FOR _idx := 0 TO RobotLibraryParameter.SUB_PROGRAM_DATA_MAX
DO
  // add command.Data[_idx]
  CreateCommandPayload.AddByte(_command.Data[_idx]);
END_FOR

// Create logging
CreateCommandPayloadLog(AxesGroup := AxesGroup);
END_METHOD

METHOD INTERNAL CreateCommandPayloadLog
VAR_IN_OUT
  /// Robot assignment of function
  AxesGroup : AxesGroup; 
END_VAR
VAR
  /// internal index for loops
 _idx : DINT;
END_VAR
// Create log entry for Parameter start
CreateLogMessage      ( Timestamp   := AxesGroup.InternalData.SystemTime,
                        MessageType := MessageType.CMD,
                        Severity    := Severity.DEBUG,
                        MessageCode := 0,
                        MessageText := 'Create command payload with the following parameter(s) :');
  
// Create log entry for EmitterID[x]
FOR _idx := 0 TO 3
DO
  CreateLogMessagePara2 ( Timestamp   := AxesGroup.InternalData.SystemTime,
                          MessageType := MessageType.CMD,
                          Severity    := Severity.DEBUG,
                          MessageCode := 0,
                          MessageText := 'Command.EmitterID[{2}] = {1}',
                          Para1       :=  SINT_TO_STRING(_command.EmitterID[_idx]),
                          Para2       :=  DINT_TO_STRING(_idx));
END_FOR

// Create log entry for ListenerID
CreateLogMessagePara1 ( Timestamp   := AxesGroup.InternalData.SystemTime,
                        MessageType := MessageType.CMD,
                        Severity    := Severity.DEBUG,
                        MessageCode := 0,
                        MessageText := 'Command.ListenerID = {1}',
                        Para1       :=  SINT_TO_STRING(_command.ListenerID));

// Create log entry for Reserve
CreateLogMessagePara1 ( Timestamp   := AxesGroup.InternalData.SystemTime,
                        MessageType := MessageType.CMD,
                        Severity    := Severity.DEBUG,
                        MessageCode := 0,
                        MessageText := 'Command.Reserve = {1}',
                        Para1       :=  BYTE_TO_STRING(_command.Reserve));

// Create log entry for JobID
CreateLogMessagePara1 ( Timestamp   := AxesGroup.InternalData.SystemTime,
                        MessageType := MessageType.CMD,
                        Severity    := Severity.DEBUG,
                        MessageCode := 0,
                        MessageText := 'Command.JobID = {1}',
                        Para1       :=  UINT_TO_STRING(_command.JobID));

FOR _idx := 0 TO RobotLibraryParameter.SUB_PROGRAM_DATA_MAX
DO
  // Create log entry for Data
  CreateLogMessagePara1 ( Timestamp   := AxesGroup.InternalData.SystemTime,
                          MessageType := MessageType.CMD,
                          Severity    := Severity.DEBUG,
                          MessageCode := 0,
                          MessageText := StrReplace('Command.Data[{0}] = {1}', '{0}', DINT_TO_STRING(_idx)), 
                          Para1       :=  UINT_TO_STRING(_command.Data[_idx]));
END_FOR
END_METHOD

METHOD FB_init : BOOL
VAR_INPUT
  /// if TRUE, the retain variables are initialized (warm start / cold start)
  bInitRetains : BOOL; 
  /// if TRUE, the instance afterwards gets moved into the copy code (online change)
  bInCopyCode  : BOOL;  
END_VAR
MyType := 'MC_CallSubprogramFB';

ExecMode := ExecutionMode.PARALLEL;
END_METHOD

METHOD PROTECTED OnCall
VAR_IN_OUT
  /// Robot assignment of function
  AxesGroup : AxesGroup; 
END_VAR
// call base implementation
SUPER^.OnCall(AxesGroup := AxesGroup);

CASE _stepCmd OF
  
  00:  IF ( _execute_R.Q )  
       THEN
         // Check function is supported and parameter are valid ?
         IF (( CheckFunctionSupported( AxesGroup := AxesGroup )) AND
             ( CheckParameterValid   ( AxesGroup := AxesGroup )))      
         THEN
           // set busy flag
           Busy := TRUE;
           // Reset command outputs
           SysDepMemSet(pDest := ADR(OutCmd), Value := 0, DataLen := SIZEOF(OutCmd));         
           // apply command parameter
          _parCmd := ParCmd;
           // init parameter sequence
          _command.ParSeq := 1;
           // create command data
           CommandData := CreateCommandPayload(AxesGroup := AxesGroup);
           // Add command to active command register
          _uniqueID := AxesGroup.Acyclic.ActiveCommandRegister.AddCmd( pCommandFB := ADR(THIS^ ));     
           // set timeout
           SetTimeout(PT := _timeoutCmd, rTimer := _timerCmd);
           // inc step counter
          _stepCmd := _stepCmd + 1; 
          END_IF
       END_IF
     

  01:  // Wait for responce received
       IF ( _responseReceived )
       THEN
         // reset response received flag
        _responseReceived := FALSE;

         CASE  _response.State 
         OF
           CmdMessageState.BUFFERED    : CommandBuffered    := TRUE;
           CmdMessageState.INTERRUPTED : CommandInterrupted := TRUE;           
           CmdMessageState.DONE        : Done               := TRUE;           
           CmdMessageState.ABORTED     : CommandAborted     := TRUE;
           CmdMessageState.ERROR       : Error              := TRUE;
         END_CASE
                
         InProgress := _response.InProgress;
         
         // Done, Aborted or Error ?
         IF (_response.State >= CmdMessageState.DONE )
         THEN
           // reset Busy flag
           Busy := FALSE;
           // Update results
           OutCmd.InstanceID        := 0; {warning 'ToDo'}
           OutCmd.OriginID          := _response.OriginID;
           OutCmd.InvocationCounter := _response.InvocationCounter;
           OutCmd.ReturnData        := _response.ReturnData;
 
           // set timeout
           SetTimeout(PT := _timeoutCmd, rTimer := _timerCmd);
           // inc step counter
          _stepCmd := _stepCmd + 1; 
         END_IF
       END_IF


  02: IF ( NOT Execute)
      THEN
        Reset();
      END_IF     
ELSE
  // invalid step
  ErrorID := RobotLibraryEvents.ERR_INVALID_STEP;
END_CASE



// Reset FB
IF ( NOT Execute )
THEN
  Reset();  
END_IF
END_METHOD

METHOD INTERNAL ParseResponsePayload : DINT
VAR_INPUT
  /// Response data
  ResponseData : RobotLibraryRecvDataFB;
  /// Timestamp
  Timestamp    : SystemTime;  
END_VAR
VAR
  /// internal index for loops
 _idx : DINT;
END_VAR

// Table 6-688: Received CMD payload (RC to PLC) of "CallSubprogram"
// --------------------------
// Header
// --------------------------
// Byte 00 : USINT   - ParSeq | State     
// Byte 01 : SINT    - AlarmMessageSeverity    
// Byte 02 : UINT    - AlarmMessageCode HB
// Byte 03 :         - AlarmMessageCode LB
// --------------------------
// Datablock
// --------------------------
// Byte 04 : USINT InvocationCounter;
// Byte 05 : SINT  Reserved;
// Byte 06 : INT   OriginID;
// Byte 07 :       OriginID;
// Byte 08 : UINT  Progress;
// Byte 09 :       Progress;
// Byte 10 : BOOL  InProgress;
// Byte 11 : BYTE  ReturnData[0];
// Byte 12 : BYTE  ReturnData[1];
// Byte 13 : BYTE  ReturnData[2];
// Byte 14 : BYTE  ReturnData[3];
// Byte 15 : BYTE  ReturnData[4];
// Byte 16 : BYTE  ReturnData[5];
// Byte 17 : BYTE  ReturnData[6];
// Byte 18 : BYTE  ReturnData[7];
// Byte 19 : BYTE  ReturnData[8];
// Byte 20 : BYTE  ReturnData[9];
// Byte 21 : BYTE  ReturnData[10];
// Byte 22 : BYTE  ReturnData[11];
// Byte 23 : BYTE  ReturnData[12];
// Byte 24 : BYTE  ReturnData[13];
// Byte 25 : BYTE  ReturnData[14];
// Byte 26 : BYTE  ReturnData[15];
// Byte 27 : BYTE  ReturnData[16];
// Byte 28 : BYTE  ReturnData[17];
// Byte 29 : BYTE  ReturnData[18];
// Byte 30 : BYTE  ReturnData[19];
// Byte 31 : BYTE  ReturnData[20];
// Byte 32 : BYTE  ReturnData[21];
// Byte 33 : BYTE  ReturnData[22];
// Byte 34 : BYTE  ReturnData[23];
// Byte 35 : BYTE  ReturnData[24];
// Byte 36 : BYTE  ReturnData[25];
// Byte 37 : BYTE  ReturnData[26];
// Byte 38 : BYTE  ReturnData[27];
// Byte 39 : BYTE  ReturnData[28];
// Byte 40 : BYTE  ReturnData[29];
// Byte 41 : BYTE  ReturnData[30];
// Byte 42 : BYTE  ReturnData[31];
// Byte 43 : BYTE  ReturnData[32];
// Byte 44 : BYTE  ReturnData[33];
// Byte 45 : BYTE  ReturnData[34];
// Byte 46 : BYTE  ReturnData[35];
// Byte 47 : BYTE  ReturnData[36];
// Byte 48 : BYTE  ReturnData[37];
// Byte 49 : BYTE  ReturnData[38];
// Byte 50 : BYTE  ReturnData[39];
// Byte 51 : BYTE  ReturnData[40];
// Byte 52 : BYTE  ReturnData[41];
// Byte 53 : BYTE  ReturnData[42];
// Byte 54 : BYTE  ReturnData[43];
// Byte 55 : BYTE  ReturnData[44];
// Byte 56 : BYTE  ReturnData[45];
// Byte 57 : BYTE  ReturnData[46];
// Byte 58 : BYTE  ReturnData[47];
// Byte 59 : BYTE  ReturnData[48];
// Byte 60 : BYTE  ReturnData[49];
// Byte 61 : BYTE  ReturnData[50];
// Byte 62 : BYTE  ReturnData[51];
// Byte 63 : BYTE  ReturnData[52];
// Byte 64 : BYTE  ReturnData[53];
// Byte 65 : BYTE  ReturnData[54];
// Byte 66 : BYTE  ReturnData[55];
// Byte 67 : BYTE  ReturnData[56];
// Byte 68 : BYTE  ReturnData[57];
// Byte 69 : BYTE  ReturnData[58];
// Byte 70 : BYTE  ReturnData[59];
// Byte 71 : BYTE  ReturnData[60];
// Byte 72 : BYTE  ReturnData[61];
// Byte 73 : BYTE  ReturnData[62];
// Byte 74 : BYTE  ReturnData[63];
// Byte 75 : BYTE  ReturnData[64];
// Byte 76 : BYTE  ReturnData[65];
// Byte 77 : BYTE  ReturnData[66];
// Byte 78 : BYTE  ReturnData[67];
// Byte 79 : BYTE  ReturnData[68];
// Byte 80 : BYTE  ReturnData[69];
// Byte 81 : BYTE  ReturnData[70];
// Byte 82 : BYTE  ReturnData[71];
// Byte 83 : BYTE  ReturnData[72];
// Byte 84 : BYTE  ReturnData[73];
// Byte 85 : BYTE  ReturnData[74];
// Byte 86 : BYTE  ReturnData[75];
// Byte 87 : BYTE  ReturnData[76];
// Byte 88 : BYTE  ReturnData[77];
// Byte 89 : BYTE  ReturnData[78];
// Byte 90 : BYTE  ReturnData[79];
// Byte 91 : BYTE  ReturnData[80];
// Byte 92 : BYTE  ReturnData[81];
// Byte 93 : BYTE  ReturnData[82];
// Byte 94 : BYTE  ReturnData[83];
// Byte 95 : BYTE  ReturnData[84];
// Byte 96 : BYTE  ReturnData[85];
// Byte 97 : BYTE  ReturnData[86];
// Byte 98 : BYTE  ReturnData[87];
// Byte 99 : BYTE  ReturnData[88];
// Byte 100: BYTE  ReturnData[89];
// Byte 101: BYTE  ReturnData[90];
// Byte 102: BYTE  ReturnData[91];
// Byte 103: BYTE  ReturnData[92];
// Byte 104: BYTE  ReturnData[93];
// Byte 105: BYTE  ReturnData[94];
// Byte 106: BYTE  ReturnData[95];
// Byte 107: BYTE  ReturnData[96];
// Byte 108: BYTE  ReturnData[97];
// Byte 109: BYTE  ReturnData[98];
// Byte 110: BYTE  ReturnData[99];
// Byte 111: BYTE  ReturnData[100];
// Byte 112: BYTE  ReturnData[101];
// Byte 113: BYTE  ReturnData[102];
// Byte 114: BYTE  ReturnData[103];
// Byte 115: BYTE  ReturnData[104];
// Byte 116: BYTE  ReturnData[105];
// Byte 117: BYTE  ReturnData[106];
// Byte 118: BYTE  ReturnData[107];
// Byte 119: BYTE  ReturnData[108];
// Byte 120: BYTE  ReturnData[109];
// Byte 121: BYTE  ReturnData[110];
// Byte 122: BYTE  ReturnData[111];
// Byte 123: BYTE  ReturnData[112];
// Byte 124: BYTE  ReturnData[113];
// Byte 125: BYTE  ReturnData[114];
// Byte 126: BYTE  ReturnData[115];
// Byte 127: BYTE  ReturnData[116];
// Byte 128: BYTE  ReturnData[117];
// Byte 129: BYTE  ReturnData[118];
// Byte 130: BYTE  ReturnData[119];
// Byte 131: BYTE  ReturnData[120];
// Byte 132: BYTE  ReturnData[121];
// Byte 133: BYTE  ReturnData[122];
// Byte 134: BYTE  ReturnData[123];
// Byte 135: BYTE  ReturnData[124];
// Byte 136: BYTE  ReturnData[125];
// Byte 137: BYTE  ReturnData[126];
// Byte 138: BYTE  ReturnData[127];
// Byte 139: BYTE  ReturnData[128];
// Byte 140: BYTE  ReturnData[129];
// Byte 141: BYTE  ReturnData[130];
// Byte 142: BYTE  ReturnData[131];
// Byte 143: BYTE  ReturnData[132];
// Byte 144: BYTE  ReturnData[133];
// Byte 145: BYTE  ReturnData[134];
// Byte 146: BYTE  ReturnData[135];
// Byte 147: BYTE  ReturnData[136];
// Byte 148: BYTE  ReturnData[137];
// Byte 149: BYTE  ReturnData[138];
// Byte 150: BYTE  ReturnData[139];
// Byte 151: BYTE  ReturnData[140];
// Byte 152: BYTE  ReturnData[141];
// Byte 153: BYTE  ReturnData[142];
// Byte 154: BYTE  ReturnData[143];
// Byte 155: BYTE  ReturnData[144];
// Byte 156: BYTE  ReturnData[145];
// Byte 157: BYTE  ReturnData[146];
// Byte 158: BYTE  ReturnData[147];
// Byte 159: BYTE  ReturnData[148];
// Byte 160: BYTE  ReturnData[149];
// Byte 161: BYTE  ReturnData[150];
// Byte 162: BYTE  ReturnData[151];
// Byte 163: BYTE  ReturnData[152];
// Byte 164: BYTE  ReturnData[153];
// Byte 165: BYTE  ReturnData[154];
// Byte 166: BYTE  ReturnData[155];
// Byte 167: BYTE  ReturnData[156];
// Byte 168: BYTE  ReturnData[157];
// Byte 169: BYTE  ReturnData[158];
// Byte 170: BYTE  ReturnData[159];
// Byte 171: BYTE  ReturnData[160];
// Byte 172: BYTE  ReturnData[161];
// Byte 173: BYTE  ReturnData[162];
// Byte 174: BYTE  ReturnData[163];
// Byte 175: BYTE  ReturnData[164];
// Byte 176: BYTE  ReturnData[165];
// Byte 177: BYTE  ReturnData[166];
// Byte 178: BYTE  ReturnData[167];
// Byte 179: BYTE  ReturnData[168];
// Byte 180: BYTE  ReturnData[169];
// Byte 181: BYTE  ReturnData[170];
// Byte 182: BYTE  ReturnData[171];
// Byte 183: BYTE  ReturnData[172];
// Byte 184: BYTE  ReturnData[173];
// Byte 185: BYTE  ReturnData[174];
// Byte 186: BYTE  ReturnData[175];
// Byte 187: BYTE  ReturnData[176];
// Byte 188: BYTE  ReturnData[177];
// Byte 189: BYTE  ReturnData[178];
// Byte 190: BYTE  ReturnData[179];
// Byte 191: BYTE  ReturnData[180];
// Byte 192: BYTE  ReturnData[181];
// Byte 193: BYTE  ReturnData[182];
// Byte 194: BYTE  ReturnData[183];
// Byte 195: BYTE  ReturnData[184];
// Byte 196: BYTE  ReturnData[185];
// Byte 197: BYTE  ReturnData[186];
// Byte 198: BYTE  ReturnData[187];
// Byte 199: BYTE  ReturnData[188];
// Byte 200: BYTE  ReturnData[189];
// call base implementation to parse the header from payload buffer
ResponseData.PayloadPtr := SUPER^.ParseResponsePayload(ResponseData := ResponseData, Timestamp := Timestamp);

// copy parsed header to response
_response.ParSeq               := _rspHeader.ParSeq;
_response.State                := _rspHeader.State;
_response.AlarmMessageSeverity := _rspHeader.AlarmMessageSeverity;
_response.AlarmMessageCode     := _rspHeader.AlarmMessageCode;

// Get Response.InvocationCounter
_response.InvocationCounter := ResponseData.GetUsint();
// Get Response.Reserve
_response.Reserve := ResponseData.GetSint();
// Get Response.OriginID
_response.OriginID := ResponseData.GetInt();
// Get Response.Progress
_response.Progress := ResponseData.GetUint();
// Get Response.InProgress
_response.InProgress := ResponseData.GetBool();

FOR _idx := 0 TO RobotLibraryParameter.SUB_PROGRAM_DATA_MAX
DO  
  // Get Response.InProgress
 _response.ReturnData[_idx] := ResponseData.GetByte();  
END_FOR

// Create logging
ParseResponsePayloadLog(ResponseData := ResponseData, Timestamp := Timestamp);
END_METHOD

METHOD INTERNAL ParseResponsePayloadLog
VAR_INPUT
  /// Response data
  ResponseData : RobotLibraryRecvDataFB;
  /// Timestamp
  Timestamp    : SystemTime;  
END_VAR
VAR
  /// internal index for loops
 _idx : DINT;
END_VAR
// Create log entry for Parameter start
CreateLogMessage      ( Timestamp   := Timestamp,
                        MessageType := MessageType.CMD,
                        Severity    := Severity.DEBUG,
                        MessageCode := 0,
                        MessageText := 'Parsed the following parameter(s) from response data:');
                        

// Create log entry for InvocationCounter
CreateLogMessagePara1 ( Timestamp   := Timestamp,
                        MessageType := MessageType.CMD,
                        Severity    := Severity.DEBUG,
                        MessageCode := 0,
                        MessageText := 'Response.InvocationCounter = {1}',
                        Para1       :=  USINT_TO_STRING(_response.InvocationCounter));

// Create log entry for Reserve
CreateLogMessagePara1 ( Timestamp   := Timestamp,
                        MessageType := MessageType.CMD,
                        Severity    := Severity.DEBUG,
                        MessageCode := 0,
                        MessageText := 'Response.Reserve = {1}',
                        Para1       :=  SINT_TO_STRING(_response.Reserve));

// Create log entry for OriginID
CreateLogMessagePara1 ( Timestamp   := Timestamp,
                        MessageType := MessageType.CMD,
                        Severity    := Severity.DEBUG,
                        MessageCode := 0,
                        MessageText := 'Response.OriginID = {1}',
                        Para1       :=  INT_TO_STRING(_response.OriginID));

// Create log entry for Progress
CreateLogMessagePara1 ( Timestamp   := Timestamp,
                        MessageType := MessageType.CMD,
                        Severity    := Severity.DEBUG,
                        MessageCode := 0,
                        MessageText := 'Response.Progress = {1}',
                        Para1       :=  UINT_TO_STRING(_response.Progress));

// Create log entry for InProgress
CreateLogMessagePara1 ( Timestamp   := Timestamp,
                        MessageType := MessageType.CMD,
                        Severity    := Severity.DEBUG,
                        MessageCode := 0,
                        MessageText := 'Response.InProgress = {1}',
                        Para1       :=  BOOL_TO_STRING(_response.InProgress));

// Create log entry for ReturnData[x]
FOR _idx := 0 TO RobotLibraryParameter.SUB_PROGRAM_DATA_MAX
DO
  CreateLogMessagePara2 ( Timestamp   := Timestamp,
                          MessageType := MessageType.CMD,
                          Severity    := Severity.DEBUG,
                          MessageCode := 0,
                          MessageText := 'Response.ReturnData[{2}] = {1}',
                          Para1       :=  BYTE_TO_STRING(_response.ReturnData[_idx]),
                          Para2       :=  DINT_TO_STRING(_idx));
END_FOR
END_METHOD

METHOD PROTECTED Reset : DINT
VAR_INPUT
END_VAR
Reset := SUPER^.Reset();

Done               := FALSE;
Busy               := FALSE;

Valid              := FALSE;
InProgress         := FALSE;
CommandAborted     := FALSE;
ParameterAccepted  := FALSE;

CommandBuffered    := FALSE;
CommandAborted     := FALSE;
CommandInterrupted := FALSE;
END_METHOD

END_FUNCTION_BLOCK

// Library/POUs/Additional/MC_CollisionDetection/MC_CollisionDetectionFB
/// Turn on/off the collision detection
FUNCTION_BLOCK MC_CollisionDetectionFB EXTENDS RobotLibraryBaseExecuteFB
// ------------------------------------------------------------------------- 
//  SRCI Robot Library                                                
// ------------------------------------------------------------------------- 
//                                                                           
//  Object:      CollisionDetectionFB                                       
//  Author:      Thorsten Brach                                                
//  Date:        2024-06-01
//
//  Description:                                              
//   
//                                                                           
//  Copyright: 
//    (C) 2024 Thorsten Brach. All rights reserved                                                                                                                                            
//             Licensed under the LGPL-3.0 license.
//                                                                           
//  Disclaimer:                                                                           
//    This project is provided without any guarantee and can be used for   
//    private and commercial purposes. Any use is at the user’s 
//    own risk and responsibility.
//
// -------------------------------------------------------------------------
VAR_INPUT
  /// Processing mode
  ProcessingMode     : ProcessingMode;
  /// Defines the target sequence in which the command will be executed
  SequenceFlag       : SequenceFlag; 
  /// Command parameter 
  ParCmd             : CollisionDetectionParCmd;
END_VAR
VAR_OUTPUT
  /// Command is transferred and confirmed by the RC
  CommandBuffered    : BOOL;
  /// The command was aborted by another command.
  CommandAborted     : BOOL;
  /// TRUE, while command is interrupted during execution and can be continued
  CommandInterrupted : BOOL;  
  /// command results
  OutCmd             : CollisionDetectionOutCmd;      
END_VAR

VAR
  /// internal copy of command parameter 
 _parCmd             : CollisionDetectionParCmd;
  /// command data to send
 _command            : CollisionDetectionSendData;
  /// response data received
 _response           : CollisionDetectionRecvData;      
END_VAR

SUPER^(AxesGroup := AxesGroup);

METHOD PROTECTED CheckFunctionSupported : BOOL
VAR_IN_OUT
  /// Robot assignment of function
  AxesGroup : AxesGroup; 
END_VAR
CheckFunctionSupported := AxesGroup.InternalData.RCSupportedFunctions.CollisionDetection;

IF ( NOT CheckFunctionSupported )
THEN
  // call base implementation for set error and create log entry
  SUPER^.CheckFunctionSupported(AxesGroup := AxesGroup);
END_IF
END_METHOD

METHOD PROTECTED CheckParameterChanged : BOOL
VAR_IN_OUT
  /// Robot assignment of function
  AxesGroup    : AxesGroup; 
END_VAR
// Check ParCmd Size is > 0, because MemCmp does not work correctly with size = 0
IF (SIZEOF(ParCmd) = 0) 
THEN 
  RETURN;
END_IF

// compare memory 
_parameterChanged := ( SysDepMemCmp(pData1 := ADR(ParCmd), pData2 := ADR(_parCmd), DataLen := SIZEOF(ParCmd)) <> RobotLibraryConstants.OK );

// check parameter valid ?
_parameterValid   := CheckParameterValid( AxesGroup := AxesGroup );

IF ((  _parameterChanged        )  AND 
    (  _parameterValid          )) OR
    (  _parameterUpdateInternal )  
THEN  
  // reset internal flag for send parameter update
 _parameterUpdateInternal := FALSE;
  // update internal copy of parameters 
 _parCmd := ParCmd;
  // inc parameter sequence
 _command.ParSeq := _command.ParSeq + 1;
  // update command data  
  CommandData := CreateCommandPayload(AxesGroup := AxesGroup); // ( Access via reference to rCommandFB in ACR )
  // notify active command register 
  AxesGroup.Acyclic.ActiveCommandRegister.NotifyParameterChanged := _uniqueID;
END_IF
END_METHOD

METHOD INTERNAL CreateCommandPayload : RobotLibrarySendDataFB
VAR_IN_OUT
  /// Robot assignment of function
  AxesGroup : AxesGroup; 
END_VAR
// Table 6-790: Sent CMD payload (PLC to RC) of "CollisionDetection"
// --------------------------
// Header
// --------------------------
// Byte 00 : UINT  - Type HB     
// Byte 01 :       - Type LB    
// Byte 02 : USINT - Reserve | ExecutionMode
// Byte 03 : USINT - ParSeq  | Priority
// --------------------------
// Datablock
// --------------------------
// Byte 04 : BOOL      - ActivateMonitoring
// Byte 05 : USINT     - UnitLimitAxis
// Byte 06 : USINT     - ThresholdMode
// Byte 07 : USINT     - ReactionMode
// Byte 08 : INT       - Sensitivity
// Byte 09 :           - Reserved
// Byte 10 : INT       - SensitivityAxis[0]
// Byte 11 :           - Reserved
// Byte 12 : INT       - SensitivityAxis[1]
// Byte 13 :           - Reserved
// Byte 14 : INT       - SensitivityAxis[2]
// Byte 15 :           - Reserved
// Byte 16 : INT       - SensitivityAxis[3]
// Byte 17 :           - Reserved
// Byte 18 : INT       - SensitivityAxis[4]
// Byte 19 :           - Reserved
// Byte 20 : INT       - SensitivityAxis[5]
// Byte 21 :           - Reserved
// Byte 22 : INT       - SensitivityAxis[6]
// Byte 23 :           - Reserved
// Byte 24 : REAL      - LimitAxis[0] HW HB
// Byte 25 :           - LimitAxis[0] HW LB
// Byte 26 :           - LimitAxis[0] LW HB
// Byte 27 :           - LimitAxis[0] LW LB
// Byte 28 : REAL      - LimitAxis[1] HW HB
// Byte 29 :           - LimitAxis[1] HW LB
// Byte 30 :           - LimitAxis[1] LW HB
// Byte 31 :           - LimitAxis[1] LW LB
// Byte 32 : REAL      - LimitAxis[2] HW HB
// Byte 33 :           - LimitAxis[2] HW LB
// Byte 34 :           - LimitAxis[2] LW HB
// Byte 35 :           - LimitAxis[2] LW LB
// Byte 36 : REAL      - LimitAxis[3] HW HB
// Byte 37 :           - LimitAxis[3] HW LB
// Byte 38 :           - LimitAxis[3] LW HB
// Byte 39 :           - LimitAxis[3] LW LB
// Byte 40 : REAL      - LimitAxis[4] HW HB
// Byte 41 :           - LimitAxis[4] HW LB
// Byte 42 :           - LimitAxis[4] LW HB
// Byte 43 :           - LimitAxis[4] LW LB
// Byte 44 : REAL      - LimitAxis[5] HW HB
// Byte 45 :           - LimitAxis[5] HW LB
// Byte 46 :           - LimitAxis[5] LW HB
// Byte 47 :           - LimitAxis[5] LW LB
// Byte 48 : REAL      - LimitAxis[6] HW HB
// Byte 49 :           - LimitAxis[6] HW LB
// Byte 50 :           - LimitAxis[6] LW HB
// Byte 51 :           - LimitAxis[6] LW LB
// --------------------------
// set command parameter 
_command.CmdTyp               :=  CmdType.CollisionDetection;
_command.ExecMode             :=  ExecMode;
_command.ParSeq               := _command.ParSeq;
_command.Priority             :=  Priority;

_command.ActivateMonitoring   := _parCmd.ActivateMonitoring;
_command.UnitLimitAxis        := _parCmd.UnitLimitAxis;
_command.ThresholdMode        := _parCmd.ThresholdMode;
_command.ReactionMode         := _parCmd.ReactionMode;
_command.Sensitivity          :=  REAL_TO_PERCENT_INT(_parCmd.Sensitivity        , IsOptional := TRUE);
_command.SensitivityAxis[0]   :=  REAL_TO_PERCENT_INT(_parCmd.SensitivityAxis[0] , IsOptional := TRUE);
_command.SensitivityAxis[1]   :=  REAL_TO_PERCENT_INT(_parCmd.SensitivityAxis[1] , IsOptional := TRUE);
_command.SensitivityAxis[2]   :=  REAL_TO_PERCENT_INT(_parCmd.SensitivityAxis[2] , IsOptional := TRUE);
_command.SensitivityAxis[3]   :=  REAL_TO_PERCENT_INT(_parCmd.SensitivityAxis[3] , IsOptional := TRUE);
_command.SensitivityAxis[4]   :=  REAL_TO_PERCENT_INT(_parCmd.SensitivityAxis[4] , IsOptional := TRUE);
_command.SensitivityAxis[5]   :=  REAL_TO_PERCENT_INT(_parCmd.SensitivityAxis[5] , IsOptional := TRUE);
_command.SensitivityAxis[6]   :=  REAL_TO_PERCENT_INT(_parCmd.SensitivityAxis[6] , IsOptional := TRUE);
_command.LimitAxis[0]         := _parCmd.LimitAxis[0];
_command.LimitAxis[1]         := _parCmd.LimitAxis[1];
_command.LimitAxis[2]         := _parCmd.LimitAxis[2];
_command.LimitAxis[3]         := _parCmd.LimitAxis[3];
_command.LimitAxis[4]         := _parCmd.LimitAxis[4];
_command.LimitAxis[5]         := _parCmd.LimitAxis[5];
_command.LimitAxis[6]         := _parCmd.LimitAxis[6];



// copy command data to header
_cmdHeader := _command;
// call base implementation to copy header to payload buffer
CreateCommandPayload := SUPER^.CreateCommandPayload(AxesGroup := AxesGroup);

// add command.ActivateMonitoring
CreateCommandPayload.AddBool(_command.ActivateMonitoring);
// add command.UnitLimitAxis
CreateCommandPayload.AddUsint(_command.UnitLimitAxis);
// add command.ThresholdMode
CreateCommandPayload.AddUsint(_command.ThresholdMode);
// add command.ReactionMode
CreateCommandPayload.AddUsint(_command.ReactionMode);
// add command.Sensitivity
CreateCommandPayload.AddInt(_command.Sensitivity);
// add command.SensitivityAxis[0]
CreateCommandPayload.AddInt(_command.SensitivityAxis[0]);
// add command.SensitivityAxis[1]
CreateCommandPayload.AddInt(_command.SensitivityAxis[1]);
// add command.SensitivityAxis[2]
CreateCommandPayload.AddInt(_command.SensitivityAxis[2]);
// add command.SensitivityAxis[3]
CreateCommandPayload.AddInt(_command.SensitivityAxis[3]);
// add command.SensitivityAxis[4]
CreateCommandPayload.AddInt(_command.SensitivityAxis[4]);
// add command.SensitivityAxis[5]
CreateCommandPayload.AddInt(_command.SensitivityAxis[5]);
// add command.SensitivityAxis[6]
CreateCommandPayload.AddInt(_command.SensitivityAxis[6]);
// add command.LimitAxis[0]
CreateCommandPayload.AddReal(_command.LimitAxis[0]);
// add command.LimitAxis[1]
CreateCommandPayload.AddReal(_command.LimitAxis[1]);
// add command.LimitAxis[2]
CreateCommandPayload.AddReal(_command.LimitAxis[2]);
// add command.LimitAxis[3]
CreateCommandPayload.AddReal(_command.LimitAxis[3]);
// add command.LimitAxis[4]
CreateCommandPayload.AddReal(_command.LimitAxis[4]);
// add command.LimitAxis[5]
CreateCommandPayload.AddReal(_command.LimitAxis[5]);
// add command.LimitAxis[6]
CreateCommandPayload.AddReal(_command.LimitAxis[6]);

// Create logging
CreateCommandPayloadLog(AxesGroup := AxesGroup);
END_METHOD

METHOD INTERNAL CreateCommandPayloadLog
VAR_IN_OUT
  /// Robot assignment of function
  AxesGroup : AxesGroup; 
END_VAR
// Create log entry for Parameter start
CreateLogMessage      ( Timestamp   := AxesGroup.InternalData.SystemTime,
                        MessageType := MessageType.CMD,
                        Severity    := Severity.DEBUG,
                        MessageCode := 0,
                        MessageText := 'Create command payload with the following parameter(s) :');
  
// Create log entry for ActivateMonitoring
CreateLogMessagePara1 ( Timestamp   := AxesGroup.InternalData.SystemTime,
                        MessageType := MessageType.CMD,
                        Severity    := Severity.DEBUG,
                        MessageCode := 0,
                        MessageText := 'Command.ActivateMonitoring = {1}',
                        Para1       :=  BOOL_TO_STRING(_command.ActivateMonitoring));

// Create log entry for UnitLimitAxis
CreateLogMessagePara1 ( Timestamp   := AxesGroup.InternalData.SystemTime,
                        MessageType := MessageType.CMD,
                        Severity    := Severity.DEBUG,
                        MessageCode := 0,
                        MessageText := 'Command.UnitLimitAxis = {1}',
                        Para1       :=  USINT_TO_STRING(_command.UnitLimitAxis));

// Create log entry for ThresholdMode
CreateLogMessagePara1 ( Timestamp   := AxesGroup.InternalData.SystemTime,
                        MessageType := MessageType.CMD,
                        Severity    := Severity.DEBUG,
                        MessageCode := 0,
                        MessageText := 'Command.ThresholdMode = {1}',
                        Para1       :=  THRESHOLD_MODE_TO_STRING(_command.ThresholdMode)); 

// Create log entry for ReactionMode
CreateLogMessagePara1 ( Timestamp   := AxesGroup.InternalData.SystemTime,
                        MessageType := MessageType.CMD,
                        Severity    := Severity.DEBUG,
                        MessageCode := 0,
                        MessageText := 'Command.ReactionMode = {1}',
                        Para1       :=  COLLISION_REACTION_MODE_TO_STRING(_command.ReactionMode)); 

// Create log entry for Sensitivity
CreateLogMessagePara1 ( Timestamp   := AxesGroup.InternalData.SystemTime,
                        MessageType := MessageType.CMD,
                        Severity    := Severity.DEBUG,
                        MessageCode := 0,
                        MessageText := 'Command.Sensitivity = {1}',
                        Para1       :=  INT_TO_STRING(_command.Sensitivity)); 

// Create log entry for SensitivityAxis[1]
CreateLogMessagePara1 ( Timestamp   := AxesGroup.InternalData.SystemTime,
                        MessageType := MessageType.CMD,
                        Severity    := Severity.DEBUG,
                        MessageCode := 0,
                        MessageText := 'Command.SensitivityAxis[1] = {1}',
                        Para1       :=  INT_TO_STRING(_command.SensitivityAxis[1]));
 
// Create log entry for SensitivityAxis[2]
CreateLogMessagePara1 ( Timestamp   := AxesGroup.InternalData.SystemTime,
                        MessageType := MessageType.CMD,
                        Severity    := Severity.DEBUG,
                        MessageCode := 0,
                        MessageText := 'Command.SensitivityAxis[2] = {1}',
                        Para1       :=  INT_TO_STRING(_command.SensitivityAxis[2]));
                        
// Create log entry for SensitivityAxis[3]
CreateLogMessagePara1 ( Timestamp   := AxesGroup.InternalData.SystemTime,
                        MessageType := MessageType.CMD,
                        Severity    := Severity.DEBUG,
                        MessageCode := 0,
                        MessageText := 'Command.SensitivityAxis[3] = {1}',
                        Para1       :=  INT_TO_STRING(_command.SensitivityAxis[3]));
                        
// Create log entry for SensitivityAxis[4]
CreateLogMessagePara1 ( Timestamp   := AxesGroup.InternalData.SystemTime,
                        MessageType := MessageType.CMD,
                        Severity    := Severity.DEBUG,
                        MessageCode := 0,
                        MessageText := 'Command.SensitivityAxis[4] = {1}',
                        Para1       :=  INT_TO_STRING(_command.SensitivityAxis[4])); 
 
// Create log entry for SensitivityAxis[5]
CreateLogMessagePara1 ( Timestamp   := AxesGroup.InternalData.SystemTime,
                        MessageType := MessageType.CMD,
                        Severity    := Severity.DEBUG,
                        MessageCode := 0,
                        MessageText := 'Command.SensitivityAxis[5] = {1}',
                        Para1       :=  INT_TO_STRING(_command.SensitivityAxis[5]));

// Create log entry for SensitivityAxis[6]
CreateLogMessagePara1 ( Timestamp   := AxesGroup.InternalData.SystemTime,
                        MessageType := MessageType.CMD,
                        Severity    := Severity.DEBUG,
                        MessageCode := 0,
                        MessageText := 'Command.SensitivityAxis[6] = {1}',
                        Para1       :=  INT_TO_STRING(_command.SensitivityAxis[6]));
                        
// Create log entry for LimitAxis[1]
CreateLogMessagePara1 ( Timestamp   := AxesGroup.InternalData.SystemTime,
                        MessageType := MessageType.CMD,
                        Severity    := Severity.DEBUG,
                        MessageCode := 0,
                        MessageText := 'Command.LimitAxis[1] = {1}',
                        Para1       :=  REAL_TO_STRING(_command.LimitAxis[1]));

// Create log entry for LimitAxis[2]
CreateLogMessagePara1 ( Timestamp   := AxesGroup.InternalData.SystemTime,
                        MessageType := MessageType.CMD,
                        Severity    := Severity.DEBUG,
                        MessageCode := 0,
                        MessageText := 'Command.LimitAxis[2] = {1}',
                        Para1       :=  REAL_TO_STRING(_command.LimitAxis[2]));
                        
// Create log entry for LimitAxis[3]
CreateLogMessagePara1 ( Timestamp   := AxesGroup.InternalData.SystemTime,
                        MessageType := MessageType.CMD,
                        Severity    := Severity.DEBUG,
                        MessageCode := 0,
                        MessageText := 'Command.LimitAxis[3] = {1}',
                        Para1       :=  REAL_TO_STRING(_command.LimitAxis[3]));
                        
// Create log entry for LimitAxis[4]
CreateLogMessagePara1 ( Timestamp   := AxesGroup.InternalData.SystemTime,
                        MessageType := MessageType.CMD,
                        Severity    := Severity.DEBUG,
                        MessageCode := 0,
                        MessageText := 'Command.LimitAxis[4] = {1}',
                        Para1       :=  REAL_TO_STRING(_command.LimitAxis[4]));

// Create log entry for LimitAxis[5]
CreateLogMessagePara1 ( Timestamp   := AxesGroup.InternalData.SystemTime,
                        MessageType := MessageType.CMD,
                        Severity    := Severity.DEBUG,
                        MessageCode := 0,
                        MessageText := 'Command.LimitAxis[5] = {1}',
                        Para1       :=  REAL_TO_STRING(_command.LimitAxis[5]));

// Create log entry for LimitAxis[6]
CreateLogMessagePara1 ( Timestamp   := AxesGroup.InternalData.SystemTime,
                        MessageType := MessageType.CMD,
                        Severity    := Severity.DEBUG,
                        MessageCode := 0,
                        MessageText := 'Command.LimitAxis[6] = {1}',
                        Para1       :=  REAL_TO_STRING(_command.LimitAxis[6]));
END_METHOD

METHOD FB_init : BOOL
VAR_INPUT
  /// if TRUE, the retain variables are initialized (warm start / cold start)
  bInitRetains : BOOL; 
  /// if TRUE, the instance afterwards gets moved into the copy code (online change)
  bInCopyCode  : BOOL;  
END_VAR
MyType := 'MC_CollisionDetectionFB';

ExecMode := ExecutionMode.PARALLEL;
END_METHOD

METHOD PROTECTED OnCall
VAR_IN_OUT
  /// Robot assignment of function
  AxesGroup : AxesGroup; 
END_VAR
// call base implementation
SUPER^.OnCall(AxesGroup := AxesGroup);

CASE _stepCmd OF
  
  00:  IF ( _execute_R.Q ) 
       THEN
         // Check function is supported and parameter are valid ?
         IF (( CheckFunctionSupported( AxesGroup := AxesGroup )) AND
             ( CheckParameterValid   ( AxesGroup := AxesGroup )))      
         THEN
           // set busy flag
           Busy := TRUE;
           // Reset command outputs
           SysDepMemSet(pDest := ADR(OutCmd), Value := 0, DataLen := SIZEOF(OutCmd));         
           // apply command parameter
          _parCmd := ParCmd;
           // init parameter sequence
          _command.ParSeq := 1;
           // create command data
           CommandData := CreateCommandPayload(AxesGroup := AxesGroup);
           // Add command to active command register
          _uniqueID := AxesGroup.Acyclic.ActiveCommandRegister.AddCmd( pCommandFB := ADR(THIS^ ));     
           // set timeout
           SetTimeout(PT := _timeoutCmd, rTimer := _timerCmd);
           // inc step counter
          _stepCmd := _stepCmd + 1; 
         END_IF
       END_IF
     

  01:  // Wait for responce received
       IF ( _responseReceived )
       THEN
         // reset response received flag
        _responseReceived := FALSE;

         CASE  _response.State 
         OF
           CmdMessageState.BUFFERED    : CommandBuffered    := TRUE;
           CmdMessageState.INTERRUPTED : CommandInterrupted := TRUE;
           CmdMessageState.DONE        : Done               := TRUE;
           CmdMessageState.ABORTED     : CommandAborted     := TRUE;
           CmdMessageState.ERROR       : Error              := TRUE;
         END_CASE
                
         // Done, Aborted or Error ?
         IF (_response.State >= CmdMessageState.DONE )
         THEN
           // Reset Busy flag
           Busy := FALSE;
           // set timeout
           SetTimeout(PT := _timeoutCmd, rTimer := _timerCmd);
           // inc step counter
          _stepCmd := _stepCmd + 1; 
         END_IF
       END_IF

  02: IF ( NOT Execute)
      THEN
        Reset();
      END_IF     
ELSE
  // invalid step
  ErrorID := RobotLibraryEvents.ERR_INVALID_STEP;
END_CASE


// Reset FB
IF ( NOT Execute )
THEN
  Reset();
END_IF
END_METHOD

METHOD INTERNAL ParseResponsePayload : DINT
VAR_INPUT
  /// Response data
  ResponseData : RobotLibraryRecvDataFB;
  /// Timestamp
  Timestamp    : SystemTime;  
END_VAR
// Table 6-791: Received CMD payload (RC to PLC) of "CollisionDetection"
// --------------------------
// Header
// --------------------------
// Byte 00 : USINT - ParSeq | State     
// Byte 01 : SINT  - AlarmMessageSeverity    
// Byte 02 : UINT  - AlarmMessageCode HB
// Byte 03 :       - AlarmMessageCode LB
// call base implementation to parse the header from payload buffer
ResponseData.PayloadPtr := SUPER^.ParseResponsePayload(ResponseData := ResponseData, Timestamp := Timestamp);

// copy parsed header to response
_response.ParSeq               := _rspHeader.ParSeq;
_response.State                := _rspHeader.State;
_response.AlarmMessageSeverity := _rspHeader.AlarmMessageSeverity;
_response.AlarmMessageCode     := _rspHeader.AlarmMessageCode;

// Create logging
ParseResponsePayloadLog(ResponseData := ResponseData, Timestamp := Timestamp);
END_METHOD

METHOD INTERNAL ParseResponsePayloadLog
VAR_INPUT
  /// Response data
  ResponseData : RobotLibraryRecvDataFB;
  /// Timestamp
  Timestamp    : SystemTime;  
END_VAR
// Create log entry for Parameter start
CreateLogMessage      ( Timestamp   := Timestamp,
                        MessageType := MessageType.CMD,
                        Severity    := Severity.DEBUG,
                        MessageCode := 0,
                        MessageText := 'Parsed the following parameter(s) from response data:');
                        
// Create log entry for no parameter 
CreateLogMessage      ( Timestamp   := Timestamp,
                        MessageType := MessageType.CMD,
                        Severity    := Severity.DEBUG,
                        MessageCode := 0,
                        MessageText := 'This command has no parameter to parse...');
END_METHOD

METHOD PROTECTED Reset : DINT
VAR_INPUT
END_VAR
Reset := SUPER^.Reset();

Done               := FALSE;
Busy               := FALSE;
CommandBuffered    := FALSE;
CommandAborted     := FALSE;
CommandInterrupted := FALSE;
END_METHOD

END_FUNCTION_BLOCK

// Library/POUs/Additional/MC_ExchangeConfiguration/MC_ExchangeConfigurationFB
/// Reads and writes specific configuration parameters on RC that are required for the RI to work
FUNCTION_BLOCK MC_ExchangeConfigurationFB EXTENDS RobotLibraryBaseEnableFB
// ------------------------------------------------------------------------- 
//  SRCI Robot Library                                                
// ------------------------------------------------------------------------- 
//                                                                           
//  Object:      ExchangeConfigurationFB                                       
//  Author:      Thorsten Brach                                                
//  Date:        2024-06-01
//
//  Description:                                              
//   
//                                                                           
//  Copyright: 
//    (C) 2024 Thorsten Brach. All rights reserved                                                                                                                                            
//             Licensed under the LGPL-3.0 license.
//                                                                           
//  Disclaimer:                                                                           
//    This project is provided without any guarantee and can be used for   
//    private and commercial purposes. Any use is at the user’s 
//    own risk and responsibility.
//
// -------------------------------------------------------------------------
VAR_INPUT
  /// Command parameter 
  ParCmd            : ExchangeConfigurationParCmd;
END_VAR

VAR_OUTPUT
  /// Command is transferred and confirmed by the RC
  CommandBuffered   : BOOL;
  /// Receiving of input parameter values has been acknowledged by RC
  ParameterAccepted : BOOL;
  /// command results
  OutCmd            : ExchangeConfigurationOutCmd;
END_VAR

VAR
  /// internal copy of command parameter 
 _parCmd            : ExchangeConfigurationParCmd;
  /// command data to send
 _command           : ExchangeConfigurationSendData;
  /// response data received
 _response          : ExchangeConfigurationRecvData;
END_VAR

SUPER^(AxesGroup := AxesGroup);

METHOD PROTECTED CheckFunctionSupported : BOOL
VAR_IN_OUT
  /// Robot assignment of function
  AxesGroup : AxesGroup; 
END_VAR
CheckFunctionSupported := AxesGroup.InternalData.RCSupportedFunctions.ExchangeConfiguration;

IF ( NOT CheckFunctionSupported )
THEN
  // call base implementation for set error and create log entry
  SUPER^.CheckFunctionSupported(AxesGroup := AxesGroup);
END_IF
END_METHOD

METHOD PROTECTED CheckParameterChanged : BOOL
VAR_IN_OUT
  /// Robot assignment of function
  AxesGroup    : AxesGroup; 
END_VAR
// Check ParCmd Size is > 0, because MemCmp does not work correctly with size = 0
IF (SIZEOF(ParCmd) = 0) 
THEN 
  RETURN;
END_IF

// compare memory 
_parameterChanged := ( SysDepMemCmp(pData1 := ADR(ParCmd), pData2 := ADR(_parCmd), DataLen := SIZEOF(ParCmd)) <> RobotLibraryConstants.OK );

// check parameter valid ?
_parameterValid   := CheckParameterValid( AxesGroup := AxesGroup );

IF ((  _parameterChanged        )  AND 
    (  _parameterValid          )) OR
    (  _parameterUpdateInternal )  
THEN  
  // reset internal flag for send parameter update
 _parameterUpdateInternal := FALSE;
  // update internal copy of parameters 
 _parCmd := ParCmd;
  // inc parameter sequence
 _command.ParSeq := _command.ParSeq + 1;
  // update command data  
  CommandData := CreateCommandPayload(AxesGroup := AxesGroup); // ( Access via reference to rCommandFB in ACR )
  // notify active command register 
  AxesGroup.Acyclic.ActiveCommandRegister.NotifyParameterChanged := _uniqueID;
  // Reset parameter accepted flag
  ParameterAccepted := FALSE;
END_IF
END_METHOD

METHOD INTERNAL CreateCommandPayload : RobotLibrarySendDataFB
VAR_IN_OUT
  /// Robot assignment of function
  AxesGroup : AxesGroup; 
END_VAR
// Table 6-86: Sent CMD payload (PLC to RC) of "ExchangeConfiguration"
// --------------------------
// Header
// --------------------------
// Byte 00 : UINT  - Type HB     
// Byte 01 :       - Type LB    
// Byte 02 : USINT - Reserve | ExecutionMode
// Byte 03 : USINT - ParSeq  | Priority
// --------------------------
// Datablock
// --------------------------
// Byte 4   : USINT      - LogLevel
// Byte 5.0 : BOOL       - WaitAtBlendingZone
// Byte 5.1 : BOOL       - Enable
// Byte 5.2 : BOOL       - AllowSecSeqWhileSubprogram
// Byte 5.3 : BOOL       - AllowDynamicBlending
// Byte 6   : UINT       - DelayTime HB
// Byte 7   :            - DelayTime LB
// Byte 8   : UINT       - WaitForNrOfCmd HB
// Byte 9   :            - WaitForNrOfCmd LB
// Byte 10  : UINT       - LifeSignTimeOut HB
// Byte 11  :            - LifeSignTimeOut LB
// Byte 12  : UINT       - SyncDelay HB
// Byte 13  :            - SyncDelay LB
// Byte 14  : USINT      - SyncReaction
// Byte 15  : DataInSync - DataInSync 
// Byte 16  : BYTE       - Reserved
// Byte 17  : BYTE       - DataEnableSync
// Byte 18  : BYTE       - Reserved
// set command parameter 
_command.CmdTyp          :=  CmdType.ExchangeConfiguration;
_command.ExecMode        :=  ExecMode;
_command.ParSeq          := _command.ParSeq;
_command.Priority        :=  Priority;
_command.LogLevel        := _parCmd.LogLevel;
_command.CtrlByte.0      := _parCmd.WaitAtBlendingZone;
_command.CtrlByte.1      :=  Enable;
_command.CtrlByte.2      := _parCmd.AllowSecSeqWhileSubprogram;
_command.CtrlByte.3      := _parCmd.AllowDynamicBlending;
_command.DelayTime       := _parCmd.DelayTime;
_command.WaitForNrOfCmd  := _parCmd.WaitForNrOfCmd;
_command.LifeSignTimeOut := _parCmd.LifeSignTimeOut;
_command.SyncDelay       := _parCmd.SyncDelay;
_command.SyncReaction    := _parCmd.SyncReaction;
_command.DataInSync      := _parCmd.DataInSync;
_command.Reserve1        := 0;
_command.DataEnableSync  := _parCmd.DataEnableSync;  
_command.Reserve2        := 0;

// copy command data to header
_cmdHeader := _command;
// call base implementation to copy header to payload buffer
CreateCommandPayload := SUPER^.CreateCommandPayload(AxesGroup := AxesGroup);

// add command.LogLevel
CreateCommandPayload.AddUsint(SINT_TO_USINT(_command.LogLevel));
// add command.CtrlByte
CreateCommandPayload.AddByte(_command.CtrlByte);
// add command.DelayTime
CreateCommandPayload.AddUint(_command.DelayTime);
// add command.WaitForNrOfCmd
CreateCommandPayload.AddUint(_command.WaitForNrOfCmd);
// add command.LifeSignTimeOut
CreateCommandPayload.AddUint(_command.LifeSignTimeOut);
// add command.SyncDelay
CreateCommandPayload.AddUint(_command.SyncDelay);
// add command.SyncReaction
CreateCommandPayload.AddUsint(_command.SyncReaction);
// add command.DataInSync
CreateCommandPayload.AddDataInSync(_command.DataInSync);
// add command.Reserve1
CreateCommandPayload.AddByte(_command.Reserve1);
// add command.DataEnableSync
CreateCommandPayload.AddDataEnableSync(_command.DataEnableSync);
// add command.Reserve2
CreateCommandPayload.AddByte(_command.Reserve2);

// Create logging
CreateCommandPayloadLog(AxesGroup := AxesGroup);
END_METHOD

METHOD INTERNAL CreateCommandPayloadLog
VAR_IN_OUT
  /// Robot assignment of function
  AxesGroup : AxesGroup; 
END_VAR
// Create log entry for Parameter start
CreateLogMessage      ( Timestamp   := AxesGroup.InternalData.SystemTime,
                        MessageType := MessageType.CMD,
                        Severity    := Severity.DEBUG,
                        MessageCode := 0,
                        MessageText := 'Create command payload with the following parameter(s) :');
  
// Create log entry for LogLevel
CreateLogMessagePara1 ( Timestamp   := AxesGroup.InternalData.SystemTime,
                        MessageType := MessageType.CMD,
                        Severity    := Severity.DEBUG,
                        MessageCode := 0,
                        MessageText := 'Command.LogLevel = {1}',
                        Para1       :=  LOG_LEVEL_TO_STRING(_command.LogLevel));

// Create log entry for CtrlByte
CreateLogMessagePara1 ( Timestamp   := AxesGroup.InternalData.SystemTime,
                        MessageType := MessageType.CMD,
                        Severity    := Severity.DEBUG,
                        MessageCode := 0,
                        MessageText := 'Command.CtrlByte = {1}',
                        Para1       :=  BYTE_TO_STRING(_command.CtrlByte));

// Create log entry for DelayTime
CreateLogMessagePara1 ( Timestamp   := AxesGroup.InternalData.SystemTime,
                        MessageType := MessageType.CMD,
                        Severity    := Severity.DEBUG,
                        MessageCode := 0,
                        MessageText := 'Command.DelayTime = {1}',
                        Para1       :=  UINT_TO_STRING(_command.DelayTime));

// Create log entry for WaitForNrOfCmd
CreateLogMessagePara1 ( Timestamp   := AxesGroup.InternalData.SystemTime,
                        MessageType := MessageType.CMD,
                        Severity    := Severity.DEBUG,
                        MessageCode := 0,
                        MessageText := 'Command.WaitForNrOfCmd = {1}',
                        Para1       :=  UINT_TO_STRING(_command.WaitForNrOfCmd));

// Create log entry for LifeSignTimeOut
CreateLogMessagePara1 ( Timestamp   := AxesGroup.InternalData.SystemTime,
                        MessageType := MessageType.CMD,
                        Severity    := Severity.DEBUG,
                        MessageCode := 0,
                        MessageText := 'Command.LifeSignTimeOut = {1}',
                        Para1       :=  UINT_TO_STRING(_command.LifeSignTimeOut));

// Create log entry for SyncDelay
CreateLogMessagePara1 ( Timestamp   := AxesGroup.InternalData.SystemTime,
                        MessageType := MessageType.CMD,
                        Severity    := Severity.DEBUG,
                        MessageCode := 0,
                        MessageText := 'Command.SyncDelay = {1}',
                        Para1       :=  UINT_TO_STRING(_command.SyncDelay));

// Create log entry for SyncReaction
CreateLogMessagePara1 ( Timestamp   := AxesGroup.InternalData.SystemTime,
                        MessageType := MessageType.CMD,
                        Severity    := Severity.DEBUG,
                        MessageCode := 0,
                        MessageText := 'Command.SyncReaction = {1}',
                        Para1       :=  SYNC_REACTION_TO_STRING(_command.SyncReaction));

// Create log entry for DataInSync
CreateLogMessagePara1 ( Timestamp   := AxesGroup.InternalData.SystemTime,
                        MessageType := MessageType.CMD,
                        Severity    := Severity.DEBUG,
                        MessageCode := 0,
                        MessageText := 'Command.DataInSync = {1}',
                        Para1       :=  DATA_IN_SYNC_TO_STRING(_command.DataInSync));

// Create log entry for Reserve1
CreateLogMessagePara1 ( Timestamp   := AxesGroup.InternalData.SystemTime,
                        MessageType := MessageType.CMD,
                        Severity    := Severity.DEBUG,
                        MessageCode := 0,
                        MessageText := 'Command.Reserve1 = {1}',
                        Para1       :=  BYTE_TO_STRING(_command.Reserve1));

// Create log entry for DataEnableSync
CreateLogMessagePara1 ( Timestamp   := AxesGroup.InternalData.SystemTime,
                        MessageType := MessageType.CMD,
                        Severity    := Severity.DEBUG,
                        MessageCode := 0,
                        MessageText := 'Command.DataEnableSync = {1}',
                        Para1       :=  DATA_ENABLE_SYNC_TO_STRING(_command.DataEnableSync));

// Create log entry for Reserve2
CreateLogMessagePara1 ( Timestamp   := AxesGroup.InternalData.SystemTime,
                        MessageType := MessageType.CMD,
                        Severity    := Severity.DEBUG,
                        MessageCode := 0,
                        MessageText := 'Command.Reserve2 = {1}',
                        Para1       :=  BYTE_TO_STRING(_command.Reserve2));
END_METHOD

METHOD FB_init : BOOL
VAR_INPUT
  /// if TRUE, the retain variables are initialized (warm start / cold start)
  bInitRetains : BOOL; 
  /// if TRUE, the instance afterwards gets moved into the copy code (online change)
  bInCopyCode  : BOOL;  
END_VAR
MyType   := 'MC_ExchangeConfigurationFB';
ExecMode := ExecutionMode.PARALLEL;
END_METHOD

METHOD PROTECTED OnCall
VAR_IN_OUT
  /// Robot assignment of function
  AxesGroup : AxesGroup; 
END_VAR
// call base implementation
SUPER^.OnCall(AxesGroup := AxesGroup);


CASE _stepCmd OF
  
  00:  IF ( _enable_R.Q ) 
       THEN
         // reset the rising edge
        _enable_R();       
         // reset the falling edge
        _enable_F();       

         // Check function is supported and parameter are valid ?
         IF (( CheckFunctionSupported( AxesGroup := AxesGroup )) AND
             ( CheckParameterValid   ( AxesGroup := AxesGroup )))      
         THEN
           // set busy flag
           Busy := TRUE;
           // Reset command outputs
           SysDepMemSet(pDest := ADR(OutCmd), Value := 0, DataLen := SIZEOF(OutCmd));         
           // apply command parameter
          _parCmd := ParCmd;
           // init parameter sequence
          _command.ParSeq := 1;
           // create command data
           CommandData := CreateCommandPayload(AxesGroup := AxesGroup);
           // Add command to active command register
          _uniqueID := AxesGroup.Acyclic.ActiveCommandRegister.AddCmd( pCommandFB := ADR(THIS^ ));     
           // set timeout
           SetTimeout(PT := _timeoutCmd, rTimer := _timerCmd);
           // inc step counter
          _stepCmd := _stepCmd + 1; 
         END_IF
       END_IF
     

  01:  // Wait for responce received
       IF ( _responseReceived )
       THEN
         // reset response received flag
        _responseReceived := FALSE;

         CASE  _response.State 
         OF
           CmdMessageState.BUFFERED    : CommandBuffered    := TRUE;
           CmdMessageState.ACTIVE      : ParameterAccepted  := TRUE;  
           CmdMessageState.ERROR       : Error              := TRUE;
         END_CASE
                
         // Active, Interrupted, Done, Aborted or Error ?
         IF (_response.State >= CmdMessageState.ACTIVE )
         THEN
           // Reset Busy Flag
           Busy := FALSE;
           // Reset Enabled flag
           Enabled := TRUE;
           
           OutCmd.LengthACR                 := _response.LengthACR;
           OutCmd.HighestToolIndex          := _response.HighestToolIndex;
           OutCmd.HighestFrameIndex         := _response.HighestFrameIndex;
           OutCmd.HighestLoadIndex          := _response.HighestLoadIndex;
           OutCmd.HighestWorkAreaIndex      := _response.HighestWorkAreaIndex;
           OutCmd.DataInSync                := _response.DataInSync;
           OutCmd.ChangeIndexTool           := _response.ChangeIndexTool;
           OutCmd.ChangeIndexFrame          := _response.ChangeIndexFrame;
           OutCmd.ChangeIndexLoad           := _response.ChangeIndexLoad;
           OutCmd.ChangeIndexWorkArea       := _response.ChangeIndexWorkArea;
           OutCmd.RAWorkingHours            := _response.RAWorkingHours;
           OutCmd.BrakeTestRequired         := _response.StatusByte.0;
           OutCmd.StepModeExactStopActive   := _response.StatusByte.1;
           OutCmd.StepModeBlendingActive    := _response.StatusByte.2;
           OutCmd.PathAccuracyMode          := _response.StatusByte.3;
           OutCmd.AvoidSingularity          := _response.StatusByte.4;
           OutCmd.CollisionDetectionEnabled := _response.StatusByte.5;
           OutCmd.AcceleratingSupported     := _response.StatusByte.6;
           OutCmd.DecceleratingSupported    := _response.StatusByte.7;
           OutCmd.ConstantVelocitySupported := _response.ConstantVelocitySupported;
           OutCmd.RCWorkingHours            := _response.RCWorkingHours;      
           // set timeout
           SetTimeout(PT := _timeoutCmd, rTimer := _timerCmd);
           // inc step counter
          _stepCmd := _stepCmd + 1; 
         END_IF
       END_IF

       // do not abort directly, so that the ParSeq update can be send
       IF ( _enable_R.Q ) OR ( _enable_F.Q ) 
       THEN
         // trigger parameter update to disable FB
        _parameterUpdateInternal := TRUE;
         // reset the rising edge
        _enable_R();       
         // reset the falling edge
        _enable_F();       
       END_IF


  02: IF (NOT Enable)
      THEN
        Reset();   
      END_IF
      
ELSE
  // invalid step
  ErrorID := RobotLibraryEvents.ERR_INVALID_STEP;
END_CASE



// Reset FB
IF (( _enable_R.Q ) OR
    ( _enable_F.Q ))
THEN
  Reset();
END_IF
END_METHOD

METHOD INTERNAL ParseResponsePayload : DINT
VAR_INPUT
  /// Response data
  ResponseData : RobotLibraryRecvDataFB;
  /// Timestamp
  Timestamp    : SystemTime;  
END_VAR
// Table 6-87: Received CMD payload (RC to PLC) of "ExchangeConfiguration"
// --------------------------
// Header
// --------------------------
// Byte 00 : USINT - ParSeq | State     
// Byte 01 : SINT  - AlarmMessageSeverity    
// Byte 02 : UINT  - AlarmMessageCode HB
// Byte 03 :       - AlarmMessageCode LB
// --------------------------
// Datablock
// --------------------------
// Byte 04 : BOOL       - Enabled
// Byte 05 : BYTE       - Reserve
// Byte 05 : UINT       - LengthACR LW HB
// Byte 06 :            - LengthACR LW LB
// Byte 08 : USINT      - HighestToolIndex
// Byte 09 : USINT      - HighestFrameIndex
// Byte 10 : USINT      - HighestLoadIndex
// Byte 11 : USINT      - HighestWorkAreaIndex
// Byte 12 : DataInSync - DataInSync
// Byte 13 : BYTE       - Reserve
// Byte 14 : USINT      - ChangeIndexTool
// Byte 15 : USINT      - ChangeIndexFrame
// Byte 16 : USINT      - ChangeIndexLoad
// Byte 17 : USINT      - ChangeIndexWorkArea
// Byte 18 : UDINT      - RA WorkingHours HW HB
// Byte 19 :            - RA WorkingHours HW LB
// Byte 20 :            - RA WorkingHours LW HB
// Byte 21 :            - RA WorkingHours LW LB
// Byte 22 : BYTE       - StatusByte
// Byte 23 : BOOL       - ConstantVelocitySupported
// Byte 24 : UDINT      - RC WorkingHours HW HB
// Byte 25 :            - RC WorkingHours HW LB
// Byte 26 :            - RC WorkingHours LW HB
// Byte 27 :            - RC WorkingHours LW LB
// --------------------------
// call base implementation to parse the header from payload buffer
ResponseData.PayloadPtr := SUPER^.ParseResponsePayload(ResponseData := ResponseData, Timestamp := Timestamp);

// copy parsed header to response
_response.ParSeq               := _rspHeader.ParSeq;
_response.State                := _rspHeader.State;
_response.AlarmMessageSeverity := _rspHeader.AlarmMessageSeverity;
_response.AlarmMessageCode     := _rspHeader.AlarmMessageCode;

// Get Response.Enabled
_response.Enabled := ResponseData.GetBool();
// Get Response.Reserve1
_response.Reserve1 := ResponseData.GetByte();
// Get Response.LengthACR
_response.LengthACR := ResponseData.GetUint();
// Get Response.HighestToolIndex
_response.HighestToolIndex := ResponseData.GetUsint();
// Get Response.HighestFrameIndex
_response.HighestFrameIndex := ResponseData.GetUsint();
// Get Response.HighestLoadIndex
_response.HighestLoadIndex := ResponseData.GetUsint();
// Get Response.HighestWorkAreaIndex
_response.HighestWorkAreaIndex := ResponseData.GetUsint();
// Get Response.DataInSync
_response.DataInSync := ResponseData.GetDataInSync();
// Get Response.Reserve2
_response.Reserve2 := ResponseData.GetByte();
// Get Response.ChangeIndexTool
_response.ChangeIndexTool := ResponseData.GetUsint();
// Get Response.ChangeIndexFrame
_response.ChangeIndexFrame := ResponseData.GetUsint();
// Get Response.ChangeIndexLoad
_response.ChangeIndexLoad := ResponseData.GetUsint();
// Get Response.ChangeIndexWorkArea
_response.ChangeIndexWorkArea := ResponseData.GetUsint();
// Get Response.RAWorkingHours
_response.RAWorkingHours := ResponseData.GetUdint();
// Get Response.StatusByte
_response.StatusByte := ResponseData.GetByte();
// Get Response.ConstantVelocitySupported
_response.ConstantVelocitySupported := ResponseData.GetBool();
// Get Response.RCWorkingHours
_response.RCWorkingHours := ResponseData.GetUdint();

// Create logging
ParseResponsePayloadLog(ResponseData := ResponseData, Timestamp := Timestamp);
END_METHOD

METHOD INTERNAL ParseResponsePayloadLog
VAR_INPUT
  /// Response data
  ResponseData : RobotLibraryRecvDataFB;
  /// Timestamp
  Timestamp    : SystemTime;  
END_VAR
// Create log entry for Parameter start
CreateLogMessage      ( Timestamp   := Timestamp,
                        MessageType := MessageType.CMD,
                        Severity    := Severity.DEBUG,
                        MessageCode := 0,
                        MessageText := 'Parsed the following parameter(s) from response data:');

// Create log entry for Enabled
CreateLogMessagePara1 ( Timestamp   := Timestamp,
                        MessageType := MessageType.CMD,
                        Severity    := Severity.DEBUG,
                        MessageCode := 0,
                        MessageText := 'Response.Enabled = {1}',
                        Para1       :=  BOOL_TO_STRING(_response.Enabled));

// Create log entry for Reserve1
CreateLogMessagePara1 ( Timestamp   := Timestamp,
                        MessageType := MessageType.CMD,
                        Severity    := Severity.DEBUG,
                        MessageCode := 0,
                        MessageText := 'Response.Reserve1 = {1}',
                        Para1       :=  BYTE_TO_STRING(_response.Reserve1));

// Create log entry for LengthACR
CreateLogMessagePara1 ( Timestamp   := Timestamp,
                        MessageType := MessageType.CMD,
                        Severity    := Severity.DEBUG,
                        MessageCode := 0,
                        MessageText := 'Response.LengthACR = {1}',
                        Para1       :=  UINT_TO_STRING(_response.LengthACR));

// Create log entry for HighestToolIndex
CreateLogMessagePara1 ( Timestamp   := Timestamp,
                        MessageType := MessageType.CMD,
                        Severity    := Severity.DEBUG,
                        MessageCode := 0,
                        MessageText := 'Response.HighestToolIndex = {1}',
                        Para1       :=  USINT_TO_STRING(_response.HighestToolIndex));

// Create log entry for HighestFrameIndex
CreateLogMessagePara1 ( Timestamp   := Timestamp,
                        MessageType := MessageType.CMD,
                        Severity    := Severity.DEBUG,
                        MessageCode := 0,
                        MessageText := 'Response.HighestFrameIndex = {1}',
                        Para1       :=  USINT_TO_STRING(_response.HighestFrameIndex));

// Create log entry for HighestLoadIndex
CreateLogMessagePara1 ( Timestamp   := Timestamp,
                        MessageType := MessageType.CMD,
                        Severity    := Severity.DEBUG,
                        MessageCode := 0,
                        MessageText := 'Response.HighestLoadIndex = {1}',
                        Para1       :=  USINT_TO_STRING(_response.HighestLoadIndex));

// Create log entry for HighestWorkAreaIndex
CreateLogMessagePara1 ( Timestamp   := Timestamp,
                        MessageType := MessageType.CMD,
                        Severity    := Severity.DEBUG,
                        MessageCode := 0,
                        MessageText := 'Response.HighestWorkAreaIndex = {1}',
                        Para1       :=  USINT_TO_STRING(_response.HighestWorkAreaIndex));

// Create log entry for DataInSync.ToolsInSync
CreateLogMessagePara1 ( Timestamp   := Timestamp,
                        MessageType := MessageType.CMD,
                        Severity    := Severity.DEBUG,
                        MessageCode := 0,
                        MessageText := 'Response.DataInSync.ToolsInSync = {1}',
                        Para1       :=  BOOL_TO_STRING(_response.DataInSync.ToolsInSync));

// Create log entry for DataInSync.FramesInSync
CreateLogMessagePara1 ( Timestamp   := Timestamp,
                        MessageType := MessageType.CMD,
                        Severity    := Severity.DEBUG,
                        MessageCode := 0,
                        MessageText := 'Response.DataInSync.FramesInSync = {1}',
                        Para1       :=  BOOL_TO_STRING(_response.DataInSync.FramesInSync));

// Create log entry for DataInSync.LoadsInSync
CreateLogMessagePara1 ( Timestamp   := Timestamp,
                        MessageType := MessageType.CMD,
                        Severity    := Severity.DEBUG,
                        MessageCode := 0,
                        MessageText := 'Response.DataInSync.LoadsInSync = {1}',
                        Para1       :=  BOOL_TO_STRING(_response.DataInSync.LoadsInSync));

// Create log entry for DataInSync.WorkAreasInSync
CreateLogMessagePara1 ( Timestamp   := Timestamp,
                        MessageType := MessageType.CMD,
                        Severity    := Severity.DEBUG,
                        MessageCode := 0,
                        MessageText := 'Response.DataInSync.WorkAreasInSync = {1}',
                        Para1       :=  BOOL_TO_STRING(_response.DataInSync.WorkAreasInSync));

// Create log entry for DataInSync.SoftwareLimitsInSync
CreateLogMessagePara1 ( Timestamp   := Timestamp,
                        MessageType := MessageType.CMD,
                        Severity    := Severity.DEBUG,
                        MessageCode := 0,
                        MessageText := 'Response.DataInSync.SoftwareLimitsInSync = {1}',
                        Para1       :=  BOOL_TO_STRING(_response.DataInSync.SoftwareLimitsInSync));
              
// Create log entry for DataInSync.DefaultDynamicsInSync
CreateLogMessagePara1 ( Timestamp   := Timestamp,
                        MessageType := MessageType.CMD,
                        Severity    := Severity.DEBUG,
                        MessageCode := 0,
                        MessageText := 'Response.DataInSync.DefaultDynamicsInSync = {1}',
                        Para1       :=  BOOL_TO_STRING(_response.DataInSync.DefaultDynamicsInSync));
               
// Create log entry for DataInSync.ReferenceDynamicsInSync
CreateLogMessagePara1 ( Timestamp   := Timestamp,
                        MessageType := MessageType.CMD,
                        Severity    := Severity.DEBUG,
                        MessageCode := 0,
                        MessageText := 'Response.DataInSync.ReferenceDynamicsInSync = {1}',
                        Para1       :=  BOOL_TO_STRING(_response.DataInSync.ReferenceDynamicsInSync));

// Create log entry for Reserve2
CreateLogMessagePara1 ( Timestamp   := Timestamp,
                        MessageType := MessageType.CMD,
                        Severity    := Severity.DEBUG,
                        MessageCode := 0,
                        MessageText := 'Response.Reserve2 = {1}',
                        Para1       :=  BYTE_TO_STRING(_response.Reserve2));

// Create log entry for ChangeIndexTool
CreateLogMessagePara1 ( Timestamp   := Timestamp,
                        MessageType := MessageType.CMD,
                        Severity    := Severity.DEBUG,
                        MessageCode := 0,
                        MessageText := 'Response.ChangeIndexTool = {1}',
                        Para1       :=  USINT_TO_STRING(_response.ChangeIndexTool));

// Create log entry for ChangeIndexFrame
CreateLogMessagePara1 ( Timestamp   := Timestamp,
                        MessageType := MessageType.CMD,
                        Severity    := Severity.DEBUG,
                        MessageCode := 0,
                        MessageText := 'Response.ChangeIndexFrame = {1}',
                        Para1       :=  USINT_TO_STRING(_response.ChangeIndexFrame));

// Create log entry for ChangeIndexLoad
CreateLogMessagePara1 ( Timestamp   := Timestamp,
                        MessageType := MessageType.CMD,
                        Severity    := Severity.DEBUG,
                        MessageCode := 0,
                        MessageText := 'Response.ChangeIndexLoad = {1}',
                        Para1       :=  USINT_TO_STRING(_response.ChangeIndexLoad));

// Create log entry for ChangeIndexWorkArea
CreateLogMessagePara1 ( Timestamp   := Timestamp,
                        MessageType := MessageType.CMD,
                        Severity    := Severity.DEBUG,
                        MessageCode := 0,
                        MessageText := 'Response.ChangeIndexWorkArea = {1}',
                        Para1       :=  USINT_TO_STRING(_response.ChangeIndexWorkArea));

// Create log entry for RAWorkingHours
CreateLogMessagePara1 ( Timestamp   := Timestamp,
                        MessageType := MessageType.CMD,
                        Severity    := Severity.DEBUG,
                        MessageCode := 0,
                        MessageText := 'Response.RAWorkingHours = {1}',
                        Para1       :=  UDINT_TO_STRING(_response.RAWorkingHours));

// Create log entry for StatusByte
CreateLogMessagePara1 ( Timestamp   := Timestamp,
                        MessageType := MessageType.CMD,
                        Severity    := Severity.DEBUG,
                        MessageCode := 0,
                        MessageText := 'Response.StatusByte = {1}',
                        Para1       :=  BYTE_TO_STRING_BIN(_response.StatusByte));

// Create log entry for ConstantVelocitySupported
CreateLogMessagePara1 ( Timestamp   := Timestamp,
                        MessageType := MessageType.CMD,
                        Severity    := Severity.DEBUG,
                        MessageCode := 0,
                        MessageText := 'Response.ConstantVelocitySupported = {1}',
                        Para1       :=  BOOL_TO_STRING(_response.ConstantVelocitySupported));

// Create log entry for RCWorkingHours
CreateLogMessagePara1 ( Timestamp   := Timestamp,
                        MessageType := MessageType.CMD,
                        Severity    := Severity.DEBUG,
                        MessageCode := 0,
                        MessageText := 'Response.RCWorkingHours = {1}',
                        Para1       :=  UDINT_TO_STRING(_response.RCWorkingHours));
END_METHOD

METHOD PROTECTED Reset : DINT
VAR_INPUT
END_VAR
Reset := SUPER^.Reset();

Busy               := FALSE;
CommandBuffered    := FALSE;
ParameterAccepted  := FALSE;
END_METHOD

END_FUNCTION_BLOCK

// Library/POUs/Additional/MC_FreeDrive/MC_FreeDriveFB
/// Move the robot axes by hand
FUNCTION_BLOCK MC_FreeDriveFB EXTENDS RobotLibraryBaseEnableFB
// ------------------------------------------------------------------------- 
//  SRCI Robot Library                                                
// ------------------------------------------------------------------------- 
//                                                                           
//  Object:      FreeDriveFB                                       
//  Author:      Thorsten Brach                                                
//  Date:        2024-06-01
//
//  Description:                                              
//   
//                                                                           
//  Copyright: 
//    (C) 2024 Thorsten Brach. All rights reserved                                                                                                                                            
//             Licensed under the LGPL-3.0 license.
//                                                                           
//  Disclaimer:                                                                           
//    This project is provided without any guarantee and can be used for   
//    private and commercial purposes. Any use is at the user’s 
//    own risk and responsibility.
//
// -------------------------------------------------------------------------
VAR_INPUT
  /// Command parameter 
  ParCmd            : FreeDriveParCmd;
END_VAR

VAR_OUTPUT
  /// Command is transferred and confirmed by the RC
  CommandBuffered   : BOOL;
  /// Receiving of input parameter values has been acknowledged by RC
  ParameterAccepted : BOOL;
  /// command results
  OutCmd            : FreeDriveOutCmd;
END_VAR

VAR
  /// internal copy of command parameter 
 _parCmd            : FreeDriveParCmd;
  /// command data to send
 _command           : FreeDriveSendData;
  /// response data received
 _response          : FreeDriveRecvData;
END_VAR

SUPER^(AxesGroup := AxesGroup);

METHOD PROTECTED CheckFunctionSupported : BOOL
VAR_IN_OUT
  /// Robot assignment of function
  AxesGroup : AxesGroup; 
END_VAR
CheckFunctionSupported := AxesGroup.InternalData.RCSupportedFunctions.FreeDrive;

IF ( NOT CheckFunctionSupported )
THEN
  // call base implementation for set error and create log entry
  SUPER^.CheckFunctionSupported(AxesGroup := AxesGroup);
END_IF
END_METHOD

METHOD PROTECTED CheckParameterChanged : BOOL
VAR_IN_OUT
  /// Robot assignment of function
  AxesGroup    : AxesGroup; 
END_VAR
// Check ParCmd Size is > 0, because MemCmp does not work correctly with size = 0
IF (SIZEOF(ParCmd) = 0) 
THEN 
  RETURN;
END_IF

// compare memory 
_parameterChanged := ( SysDepMemCmp(pData1 := ADR(ParCmd), pData2 := ADR(_parCmd), DataLen := SIZEOF(ParCmd)) <> RobotLibraryConstants.OK );

// check parameter valid ?
_parameterValid   := CheckParameterValid( AxesGroup := AxesGroup );

IF ((  _parameterChanged        )  AND 
    (  _parameterValid          )) OR
    (  _parameterUpdateInternal )  
THEN  
  // reset internal flag for send parameter update
 _parameterUpdateInternal := FALSE;
  // update internal copy of parameters 
 _parCmd := ParCmd;
  // inc parameter sequence
 _command.ParSeq := _command.ParSeq + 1;
  // update command data  
  CommandData := CreateCommandPayload(AxesGroup := AxesGroup); // ( Access via reference to rCommandFB in ACR )
  // notify active command register 
  AxesGroup.Acyclic.ActiveCommandRegister.NotifyParameterChanged := _uniqueID;
  // Reset parameter accepted flag
  ParameterAccepted := FALSE;
END_IF
END_METHOD

METHOD INTERNAL CreateCommandPayload : RobotLibrarySendDataFB
VAR_IN_OUT
  /// Robot assignment of function
  AxesGroup : AxesGroup; 
END_VAR
// Table 6-797: Sent CMD payload (PLC to RC) of "FreeDrive"
// --------------------------
// Header
// --------------------------
// Byte 00 : UINT  - Type HB     
// Byte 01 :       - Type LB    
// Byte 02 : USINT - Reserve | ExecutionMode
// Byte 03 : USINT - ParSeq  | Priority
// --------------------------
// Datablock
// --------------------------
// Byte 4  : BOOL  - Enable
// set command parameter 
_command.CmdTyp     :=  CmdType.FreeDrive;
_command.ExecMode   :=  ExecMode;
_command.ParSeq     := _command.ParSeq;
_command.Priority   :=  Priority;
_command.Enable     := Enable;

// copy command data to header
_cmdHeader := _command;
// call base implementation to copy header to payload buffer
CreateCommandPayload := SUPER^.CreateCommandPayload(AxesGroup := AxesGroup);

// add command.Enable
CreateCommandPayload.AddBool(_command.Enable);

// Create logging
CreateCommandPayloadLog(AxesGroup := AxesGroup);
END_METHOD

METHOD INTERNAL CreateCommandPayloadLog
VAR_IN_OUT
  /// Robot assignment of function
  AxesGroup : AxesGroup; 
END_VAR
// Create log entry for Parameter start
CreateLogMessage      ( Timestamp   := AxesGroup.InternalData.SystemTime,
                        MessageType := MessageType.CMD,
                        Severity    := Severity.DEBUG,
                        MessageCode := 0,
                        MessageText := 'Create command payload with the following parameter(s) :');
  
// Create log entry for Enable
CreateLogMessagePara1 ( Timestamp   := AxesGroup.InternalData.SystemTime,
                        MessageType := MessageType.CMD,
                        Severity    := Severity.DEBUG,
                        MessageCode := 0,
                        MessageText := 'Command.Enable = {1}',
                        Para1       :=  BOOL_TO_STRING(_command.Enable));
END_METHOD

METHOD FB_init : BOOL
VAR_INPUT
  /// if TRUE, the retain variables are initialized (warm start / cold start)
  bInitRetains : BOOL; 
  /// if TRUE, the instance afterwards gets moved into the copy code (online change)
  bInCopyCode  : BOOL;  
END_VAR
MyType := 'MC_FreeDriveFB';
END_METHOD

METHOD PROTECTED OnCall
VAR_IN_OUT
  /// Robot assignment of function
  AxesGroup : AxesGroup; 
END_VAR
// call base implementation
SUPER^.OnCall(AxesGroup := AxesGroup);

CASE _stepCmd OF
  
  00:  IF ( _enable_R.Q ) 
       THEN
         // reset the rising edge
        _enable_R();       
         // reset the falling edge
        _enable_F();    
 
         // Check function is supported and parameter are valid ?
         IF (( CheckFunctionSupported( AxesGroup := AxesGroup )) AND
             ( CheckParameterValid   ( AxesGroup := AxesGroup )))      
         THEN
           // set busy flag
           Busy := TRUE;
           // Reset command outputs
           SysDepMemSet(pDest := ADR(OutCmd), Value := 0, DataLen := SIZEOF(OutCmd));         
           // apply command parameter
          _parCmd := ParCmd;
           // init parameter sequence
          _command.ParSeq := 1;
           // create command data
           CommandData := CreateCommandPayload(AxesGroup := AxesGroup);
           // Add command to active command register
          _uniqueID := AxesGroup.Acyclic.ActiveCommandRegister.AddCmd( pCommandFB := ADR(THIS^ ));     
           // set timeout
           SetTimeout(PT := _timeoutCmd, rTimer := _timerCmd);
           // inc step counter
          _stepCmd := _stepCmd + 1; 
         END_IF
       END_IF
 
    
  01:  // Wait for responce received
       IF ( _responseReceived )
       THEN
         // reset response received flag
        _responseReceived := FALSE;

         CASE  _response.State 
         OF
           CmdMessageState.BUFFERED    : CommandBuffered    := TRUE;
           CmdMessageState.ACTIVE      : ParameterAccepted  := TRUE;           
           CmdMessageState.ERROR       : Error              := TRUE;
         END_CASE
         
         // Update results
         OutCmd.Enabled := _response.Enabled;
                
         // Done, Aborted or Error ?
         IF (_response.State >= CmdMessageState.DONE )
         THEN
           // Reset Enabled flag
           Enabled := FALSE;
           // set timeout
           SetTimeout(PT := _timeoutCmd, rTimer := _timerCmd);
           // inc step counter
          _stepCmd := _stepCmd + 1; 
         END_IF
       END_IF
       
       // do not abort directly, so that the ParSeq update can be send
       IF ( _enable_R.Q ) OR ( _enable_F.Q ) 
       THEN
         // trigger parameter update to disable FB
        _parameterUpdateInternal := TRUE;
         // reset the rising edge
        _enable_R();       
         // reset the falling edge
        _enable_F();       
       END_IF


  02: IF (NOT Enable)
      THEN
        Reset();   
      END_IF
      
ELSE
  // invalid step
  ErrorID := RobotLibraryEvents.ERR_INVALID_STEP;
END_CASE



// Reset FB
IF (( _enable_R.Q ) OR
    ( _enable_F.Q ))
THEN
  Reset();
END_IF
END_METHOD

METHOD INTERNAL ParseResponsePayload : DINT
VAR_INPUT
  /// Response data
  ResponseData : RobotLibraryRecvDataFB;
  /// Timestamp
  Timestamp    : SystemTime;  
END_VAR
// Table 6-798: Received CMD payload (RC to PLC) of "FreeDrive"
// --------------------------
// Header
// --------------------------
// Byte 00 : USINT - ParSeq | State     
// Byte 01 : SINT  - AlarmMessageSeverity    
// Byte 02 : UINT  - AlarmMessageCode HB
// Byte 03 :       - AlarmMessageCode LB
// --------------------------
// Datablock
// --------------------------
// Byte 04 : BOOL       - Enabled
// --------------------------
// call base implementation to parse the header from payload buffer
ResponseData.PayloadPtr := SUPER^.ParseResponsePayload(ResponseData := ResponseData, Timestamp := Timestamp);

// copy parsed header to response
_response.ParSeq               := _rspHeader.ParSeq;
_response.State                := _rspHeader.State;
_response.AlarmMessageSeverity := _rspHeader.AlarmMessageSeverity;
_response.AlarmMessageCode     := _rspHeader.AlarmMessageCode;

// Get Response.Enabled
_response.Enabled := ResponseData.GetBool();

// Create logging
ParseResponsePayloadLog(ResponseData := ResponseData, Timestamp := Timestamp);
END_METHOD

METHOD INTERNAL ParseResponsePayloadLog
VAR_INPUT
  /// Response data
  ResponseData : RobotLibraryRecvDataFB;
  /// Timestamp
  Timestamp    : SystemTime;  
END_VAR
// Create log entry for Parameter start
CreateLogMessage      ( Timestamp   := Timestamp,
                        MessageType := MessageType.CMD,
                        Severity    := Severity.DEBUG,
                        MessageCode := 0,
                        MessageText := 'Parsed the following parameter(s) from response data:');
                        
// Create log entry for Enabled
CreateLogMessagePara1 ( Timestamp   := Timestamp,
                        MessageType := MessageType.CMD,
                        Severity    := Severity.DEBUG,
                        MessageCode := 0,
                        MessageText := 'Response.Enabled = {1}',
                        Para1       :=  BOOL_TO_STRING(_response.Enabled));
END_METHOD

METHOD PROTECTED Reset : DINT
VAR_INPUT
END_VAR
Reset := SUPER^.Reset();

Busy               := FALSE;
CommandBuffered    := FALSE;
ParameterAccepted  := FALSE;
END_METHOD

END_FUNCTION_BLOCK

// Library/POUs/Additional/MC_MeasuringInput/MC_MeasuringInputFB
/// Capture trigger Position, measuring input
FUNCTION_BLOCK MC_MeasuringInputFB EXTENDS RobotLibraryBaseExecuteFB
// ------------------------------------------------------------------------- 
//  SRCI Robot Library                                                
// ------------------------------------------------------------------------- 
//                                                                           
//  Object:      MeasuringInputFB                                       
//  Author:      Thorsten Brach                                                
//  Date:        2024-06-01
//
//  Description:                                              
//   
//                                                                           
//  Copyright: 
//    (C) 2024 Thorsten Brach. All rights reserved                                                                                                                                            
//             Licensed under the LGPL-3.0 license.
//                                                                           
//  Disclaimer:                                                                           
//    This project is provided without any guarantee and can be used for   
//    private and commercial purposes. Any use is at the user’s 
//    own risk and responsibility.
//
// -------------------------------------------------------------------------
VAR_INPUT
  /// Command parameter 
  ParCmd          : MeasuringInputParCmd;        
END_VAR

VAR_OUTPUT
  /// Command is transferred and confirmed by the RC
  CommandBuffered : BOOL;  
  /// Command output 
  OutCmd          : MeasuringInputOutCmd;            
END_VAR
VAR
  /// internal copy of command parameter 
 _parCmd          : MeasuringInputParCmd;
  /// command data to send
 _command         : MeasuringInputSendData;
  /// response data received
 _response        : MeasuringInputRecvData;      
END_VAR

SUPER^(AxesGroup := AxesGroup);

METHOD PROTECTED CheckFunctionSupported : BOOL
VAR_IN_OUT
  /// Robot assignment of function
  AxesGroup : AxesGroup; 
END_VAR
CheckFunctionSupported := AxesGroup.InternalData.RCSupportedFunctions.MeasuringInput;

IF ( NOT CheckFunctionSupported )
THEN
  // call base implementation for set error and create log entry
  SUPER^.CheckFunctionSupported(AxesGroup := AxesGroup);
END_IF
END_METHOD

METHOD PROTECTED CheckParameterChanged : BOOL
VAR_IN_OUT
  /// Robot assignment of function
  AxesGroup    : AxesGroup; 
END_VAR
// Check ParCmd Size is > 0, because MemCmp does not work correctly with size = 0
IF (SIZEOF(ParCmd) = 0) 
THEN 
  RETURN;
END_IF

// compare memory 
_parameterChanged := ( SysDepMemCmp(pData1 := ADR(ParCmd), pData2 := ADR(_parCmd), DataLen := SIZEOF(ParCmd)) <> RobotLibraryConstants.OK );

// check parameter valid ?
_parameterValid   := CheckParameterValid( AxesGroup := AxesGroup );

IF ((  _parameterChanged        )  AND 
    (  _parameterValid          )) OR
    (  _parameterUpdateInternal )  
THEN  
  // reset internal flag for send parameter update
 _parameterUpdateInternal := FALSE;
  // update internal copy of parameters 
 _parCmd := ParCmd;
  // inc parameter sequence
 _command.ParSeq := _command.ParSeq + 1;
  // update command data  
  CommandData := CreateCommandPayload(AxesGroup := AxesGroup); // ( Access via reference to rCommandFB in ACR )
  // notify active command register 
  AxesGroup.Acyclic.ActiveCommandRegister.NotifyParameterChanged := _uniqueID;
END_IF
END_METHOD

METHOD INTERNAL CreateCommandPayload : RobotLibrarySendDataFB
VAR_IN_OUT
  /// Robot assignment of function
  AxesGroup : AxesGroup; 
END_VAR
// Table 6-565: Sent CMD payload (PLC to RC) of "MeasuringInput"
// --------------------------
// Header
// --------------------------
// Byte 000 : UINT  - Type HB     
// Byte 001 :       - Type LB    
// Byte 002 : USINT - Reserve | ExecutionMode
// Byte 003 : USINT - ParSeq  | Priority
// --------------------------
// Datablock
// --------------------------
// Byte 004 : USINT       - MeasuringMode
// Byte 005 : USINT       - Index
// Byte 006 : USINT       - BitNumber
// set command parameter 
_command.CmdTyp        :=  CmdType.MeasuringInput;
_command.ExecMode      :=  ExecMode;
_command.ParSeq        := _command.ParSeq;
_command.Priority      :=  Priority;
                       
_command.MeasuringMode := parCmd.MeasuringMode;
_command.Index         := parCmd.Index;
_command.BitNumber     := parCmd.BitNumber;

// copy command data to header
_cmdHeader := _command;
// call base implementation to copy header to payload buffer
CreateCommandPayload := SUPER^.CreateCommandPayload(AxesGroup := AxesGroup);

// add command.MeasuringMode
CreateCommandPayload.AddUsint(_command.MeasuringMode);
// add command.Index
CreateCommandPayload.AddUsint(_command.Index);
// add command.BitNumber
CreateCommandPayload.AddUsint(_command.BitNumber);

// Create logging
CreateCommandPayloadLog(AxesGroup := AxesGroup);
END_METHOD

METHOD INTERNAL CreateCommandPayloadLog
VAR_IN_OUT
  /// Robot assignment of function
  AxesGroup : AxesGroup; 
END_VAR
// Create log entry for Parameter start
CreateLogMessage      ( Timestamp   := AxesGroup.InternalData.SystemTime,
                        MessageType := MessageType.CMD,
                        Severity    := Severity.DEBUG,
                        MessageCode := 0,
                        MessageText := 'Create command payload with the following parameter(s) :');
  
// Create log entry for MeasuringMode
CreateLogMessagePara1 ( Timestamp   := AxesGroup.InternalData.SystemTime,
                        MessageType := MessageType.CMD,
                        Severity    := Severity.DEBUG,
                        MessageCode := 0,
                        MessageText := 'Command.MeasuringMode = {1}',
                        Para1       :=  USINT_TO_STRING(_command.MeasuringMode));
                        
// Create log entry for Index
CreateLogMessagePara1 ( Timestamp   := AxesGroup.InternalData.SystemTime,
                        MessageType := MessageType.CMD,
                        Severity    := Severity.DEBUG,
                        MessageCode := 0,
                        MessageText := 'Command.Index = {1}',
                        Para1       :=  USINT_TO_STRING(_command.Index));
                        
// Create log entry for BitNumber
CreateLogMessagePara1 ( Timestamp   := AxesGroup.InternalData.SystemTime,
                        MessageType := MessageType.CMD,
                        Severity    := Severity.DEBUG,
                        MessageCode := 0,
                        MessageText := 'Command.BitNumber = {1}',
                        Para1       :=  USINT_TO_STRING(_command.BitNumber));
END_METHOD

METHOD FB_init : BOOL
VAR_INPUT
  /// if TRUE, the retain variables are initialized (warm start / cold start)
  bInitRetains : BOOL; 
  /// if TRUE, the instance afterwards gets moved into the copy code (online change)
  bInCopyCode  : BOOL;  
END_VAR
MyType := 'MC_MeasuringInputFB';

ExecMode := ExecutionMode.PARALLEL;
END_METHOD

METHOD PROTECTED OnCall
VAR_IN_OUT
  /// Robot assignment of function
  AxesGroup : AxesGroup; 
END_VAR
// call base implementation
SUPER^.OnCall(AxesGroup := AxesGroup);

CASE _stepCmd OF
  
  00:  IF ( _execute_R.Q )  
       THEN
         // Check function is supported and parameter are valid ?
         IF (( CheckFunctionSupported( AxesGroup := AxesGroup )) AND
             ( CheckParameterValid   ( AxesGroup := AxesGroup )))      
         THEN
           // set busy flag
           Busy := TRUE;
           // Reset command outputs
           SysDepMemSet(pDest := ADR(OutCmd), Value := 0, DataLen := SIZEOF(OutCmd));         
           // apply command parameter
          _parCmd := ParCmd;
           // init parameter sequence
          _command.ParSeq := 1;
           // create command data
           CommandData := CreateCommandPayload(AxesGroup := AxesGroup);
           // Add command to active command register
          _uniqueID := AxesGroup.Acyclic.ActiveCommandRegister.AddCmd( pCommandFB := ADR(THIS^ ));     
           // set timeout
           SetTimeout(PT := _timeoutCmd, rTimer := _timerCmd);
           // inc step counter
          _stepCmd := _stepCmd + 1;
         END_IF 
       END_IF
     

  01:  // Wait for responce received
       IF ( _responseReceived )
       THEN
         // reset response received flag
        _responseReceived := FALSE;

         CASE  _response.State 
         OF
           CmdMessageState.BUFFERED    : CommandBuffered := TRUE;
           CmdMessageState.DONE        : Done            := TRUE;
           CmdMessageState.ERROR       : Error           := TRUE;
         END_CASE
                
         // Done, Aborted or Error ?
         IF (_response.State >= CmdMessageState.DONE )
         THEN
           // Reset Busy flag
           Busy := FALSE;
           // Update results
           OutCmd.MeasuringID := _response.MeasuringID;
           OutCmd.Measurings  := _response.Measurings;
           
           // set timeout
           SetTimeout(PT := _timeoutCmd, rTimer := _timerCmd);
           // inc step counter
          _stepCmd := _stepCmd + 1; 
         END_IF
       END_IF

  02: IF ( NOT Execute)
      THEN
        Reset();
      END_IF     
ELSE
  // invalid step
  ErrorID := RobotLibraryEvents.ERR_INVALID_STEP;
END_CASE



// Reset FB
IF ( NOT Execute )
THEN
  Reset();  
END_IF
END_METHOD

